(* Schneider Machine Expert - Basic project trying comparison block, file version 2.7.0.0 *)
(* ProjectInformations: Name=New project *)

HARDWARE
  Cpu 0: TM221M16R/G
  EthernetConfiguration: NetworkName=M221, IpAllocationMode=FixedAddress, IpAddress=0.0.0.0, SubnetMask=0.0.0.0
  SerialLineConfiguration: Baud=Baud19200, Parity=ParityEven, DataBits=DataBits8, StopBits=StopBits1, PhysicalMedium=PhysicalMediumRs485, TransmissionMode=TransmissionModeModbusRtu, SlaveId=1, Addressing=SlaveAddressing
  MastTask: UsePeriodScanMode=false, PeriodScan=100
  FastTask: Period=255
  CpuBehavior: StartingMode=StartAsPreviousState, AutoSaveRamOnEeprom=true, WatchdogPeriod=250

SYMBOLS  (address, symbol, comment, settings)
  %MW0      VAR_A
  %MW1      VAR_B
  %MW2      VAR_C
  %MW3      VAR_D
  %MW4      A_SMALLER_THAN_B
  %Q0.0     LAMP

POU New POU
  (* SectionNumber=1 *)

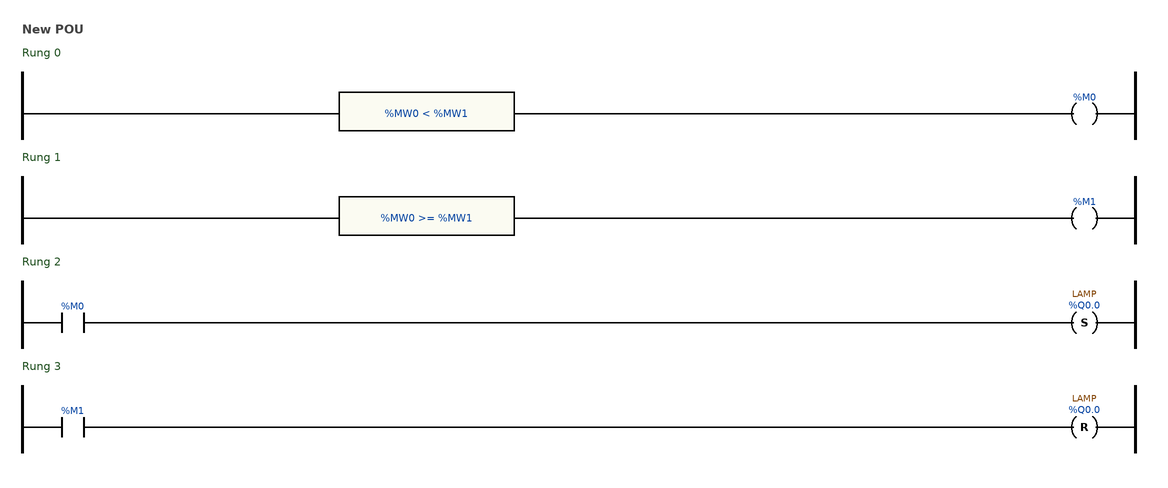

// Rung 0
  LD [ %MW0 < %MW1 ]      (* VAR_A, VAR_B *)
  ST %M0
  // as ST:
  //   %M0 := VAR_A < VAR_B;

// Rung 1
  LD 1
  AND [ %MW0 >= %MW1 ]    (* VAR_A, VAR_B *)
  ST %M1
  // as ST:
  //   %M1 := VAR_A >= VAR_B;

// Rung 2
  LD %M0
  S %Q0.0                 (* LAMP *)
  // as ST:
  //   IF %M0 THEN LAMP := TRUE; END_IF;

// Rung 3
  LD %M1
  R %Q0.0                 (* LAMP *)
  // as ST:
  //   IF %M1 THEN LAMP := FALSE; END_IF;
